// TIA Portal V19 export
TYPE "UDT_ALARMACKN"
   STRUCT
      setup : Struct   // HMI Setup
         en { S7_SetPoint := 'True'} : Bool := false;   // Enable alarm
         spon { S7_SetPoint := 'True'} : Real := 0.0;   // Setpoint for delay on timer (Real number because we count every 100ms)
      END_STRUCT;
      don : Struct   // Delay on for alarming
         countup : Bool := false;   // Command to start counting
         sp : UInt := 0;   // SP in x100ms
         actual : UInt := 0;   // Actual time elapsed
         end : Bool := false;   // End of measurement
      END_STRUCT;
      status : Struct   // Status
         plcackn : Bool := false;   // PLC acknowledgement
         alarm : Bool := false;   // Alarm
         siren : Bool := false;   // Siren
      END_STRUCT;
   END_STRUCT;
END_TYPE
